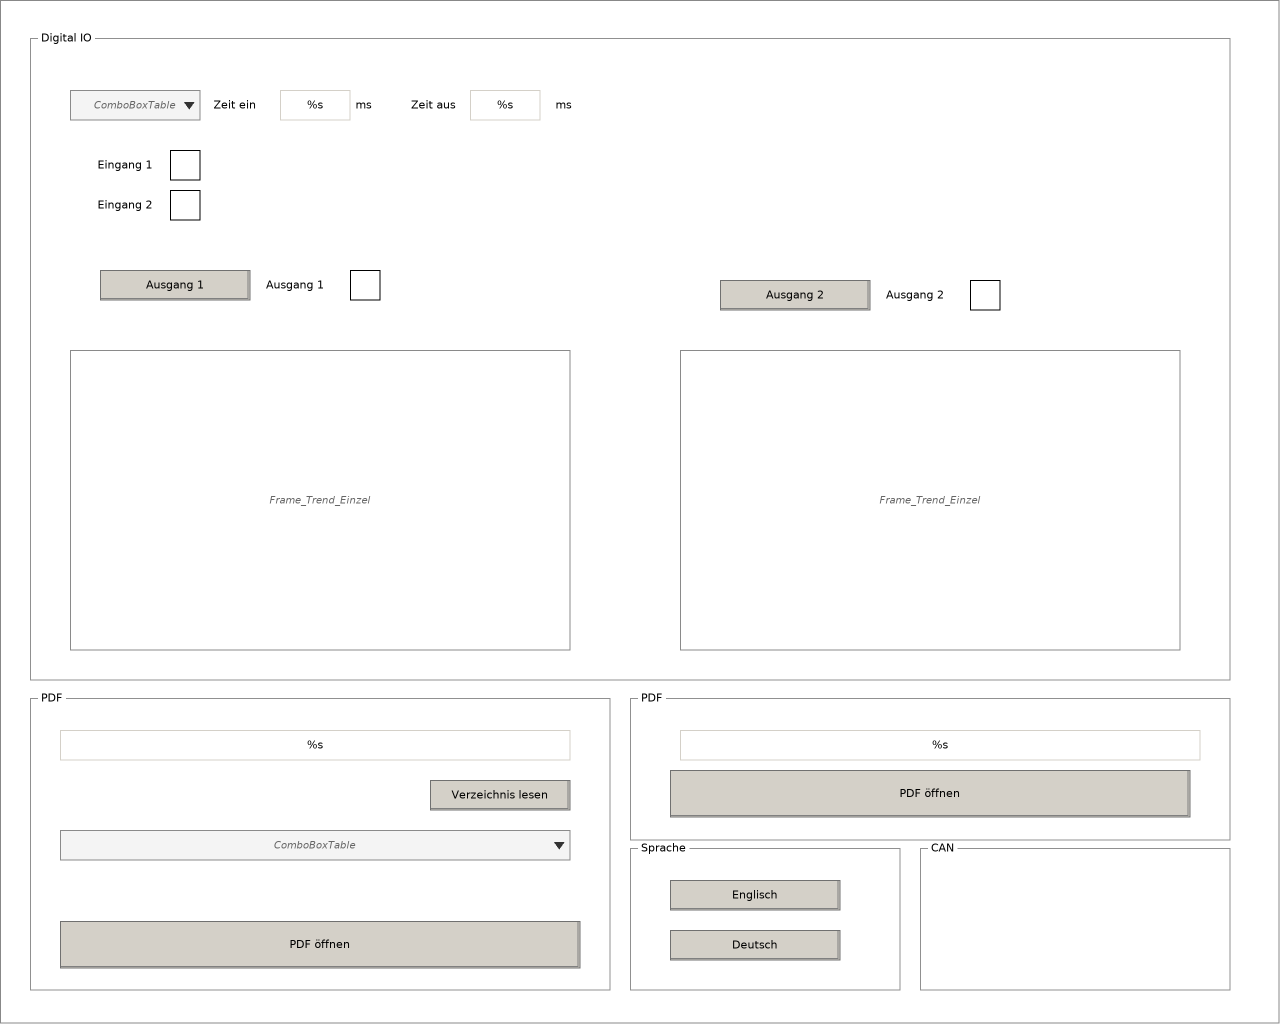
VISUALIZATION Visualization  // 1280x1024
    GroupBox (30,30 1200x650), "Digital IO"
        Rectangle (320,240 30x30), colour toggle: MAIN.ATQ_output1
        Rectangle (140,120 30x30), colour toggle: MAIN.ATI_input1
        Rectangle (140,160 30x30), colour toggle: MAIN.ATI_input2
        Rectangle (940,250 30x30), colour toggle: MAIN.ATQ_output2
        Label (40,120 110x30), "Eingang 1"
        Label (160,60 90x30), "Zeit ein"
        Label (830,250 110x30), "Ausgang 2"
        Label (210,240 110x30), "Ausgang 1"
        Button (690,250 150x30), "Ausgang 2"
            toggle MAIN.ATQ_output2
        Button (70,240 150x30), "Ausgang 1"
            toggle MAIN.ATQ_output1
        Textfield (440,60 70x30), "%s", text variable: MAIN.szeit_off
            OnMouseClick: write the text variable via Default
        Textfield (250,60 70x30), "%s", text variable: MAIN.szeit_on
            OnMouseClick: write the text variable via Default
        Label (40,160 110x30), "Eingang 2"
        Label (360,60 90x30), "Zeit aus"
        Label (320,60 27x30), "ms"
        ComboBoxTable (40,60 130x30), variable: Main.auswahl_index, data array: MAIN.auswahl
            p3854506369: MAIN.auswahl[INDEX]
        Label (520,60 27x30), "ms"
        Frame (650,320 500x300)
            shows Frame_Trend_Einzel(itemValue := PRG_Visualisierung.fbpwmTrend[2].itemValue)
        Frame (40,320 500x300)
            shows Frame_Trend_Einzel(itemValue := PRG_Visualisierung.fbpwmTrend[1].itemValue)
    GroupBox (920,840 310x150), "CAN"
    GroupBox (630,840 270x150), "Sprache"
        Button (40,40 170x30), "Englisch"
            OnMouseClick: ChangeLanguage ChangeLanguage=EN
        Button (40,90 170x30), "Deutsch"
            OnMouseClick: ChangeLanguage ChangeLanguage=DE
    GroupBox (30,690 580x300), "PDF"
        Button (400,90 140x30), "Verzeichnis lesen"
            tap MAIN.ctrl_readdir.Execute
        Textfield (30,40 510x30), "%s", text variable: MAIN.Pfadname
            OnMouseClick: write the text variable via Default
        ComboBoxTable (30,140 510x30), variable: MAIN.dateiindex, data array: MAIN.fbdirectoryRead.List
            p1892666644: MAIN.fbdirectoryRead.fbEnumFindFileList.sPathName
            p338671338: MAIN.fbdirectoryRead.fbEnumFindFileList.eCmd
            p2170511999: MAIN.fbdirectoryRead.fbEnumFindFileList.pFindList^
            p3723444502: MAIN.fbdirectoryRead.fbEnumFindFileList.cbFindList
            p1218418051: MAIN.fbdirectoryRead.fbEnumFindFileList.bExecute
            p746581629: MAIN.fbdirectoryRead.fbEnumFindFileList.tTimeout
            p3104783080: MAIN.fbdirectoryRead.fbEnumFindFileList.bBusy
            p2501879983: MAIN.fbdirectoryRead.fbEnumFindFileList.bError
            p7306298: MAIN.fbdirectoryRead.fbEnumFindFileList.nErrID
            p1933151965: MAIN.fbdirectoryRead.fbEnumFindFileList.bEOE
            p3863566920: MAIN.fbdirectoryRead.fbEnumFindFileList.nFindFiles
            p2192122294: MAIN.fbdirectoryRead.fbEnumFindFileList.fbEnum
            p400160035: MAIN.fbdirectoryRead.fbEnumFindFileList.fbTrigger
            p1265227338: MAIN.fbdirectoryRead.fbEnumFindFileList.state
            p3726181087: MAIN.fbdirectoryRead.fbEnumFindFileList.cbEntry
            p3136911649: MAIN.fbdirectoryRead.fbEnumFindFileList.nEntries
            p797552052: MAIN.fbdirectoryRead.fbEnumFindFileList.pEntry^
            p3854506369: MAIN.fbdirectoryRead.List[INDEX]
        Button (30,231 520x47), "PDF öffnen"
            tap MAIN.ctrl_pdf_2.Execute
    GroupBox (630,690 600x150), "PDF"
        Button (40,80 520x47), "PDF öffnen"
            tap MAIN.ctrl_pdf_1.Execute
        Textfield (50,40 520x30), "%s", text variable: MAIN.dateiname
            OnMouseClick: write the text variable via Default
END_VISUALIZATION

(* stored: Version 1.1.0.1, ProductVersion 3.1.4020.12
   Visu Visualization: Id {a301f14c-5bc0-4aa7-85f4-2f75619349cc} *)
